// TIA Portal V19 export
TYPE "LAF_typeAxisDiagUnits"
TITLE = LAF_typeAxisDiagUnits
// Length and velocity units of a Technology Object
// stored: Access Published
   STRUCT
      lengthUnit { ExternalWritable := 'False'} : UDInt;   // Unit for position (1004=rad, 1005=°, 1010=m, 1011=km, 1013=mm, 1014=µm, 1015=nm, 1018=ft, 1019=in, 1021=mi); with high resolution (1536=mm, 1537=°)
      velocityUnit { ExternalWritable := 'False'} : UDInt;   // Unit for velocity (1061=m/s, 1062=mm/s, 1063=m/h 1064=km/h, 1066=in/s, 1067=ft/s, 1069=in/min, 1070=ft/min, 1075=mi/h, 1082=1/s, 1083=1/min, 1086=rad/s, 1521=°/s, 1522=°/min, 1523=rad/min, 1524=mm/min, 1525=m/min, 1526=mm/h, 1527=km/min, 1528=1/h); with high resolution (1538=mm/s, 1539=°/s) / Unit for velocity (1061=m/s, 1062=mm/s, 1063=m/h 1064=km/h, 1066=in/s, 1067=ft/s, 1069=in/min, 1070=ft/min, 1075=mi/h, 1082=1/s, 1083=1/min, 1086=rad/s, 1521=°/s, 1522=°/min, 1523=rad/min=1524: mm/min, 1525=m/min, 1526=mm/h, 1527=km/min, 1528=1/h); with high resolution (1538=mm/s, 1539=°/s)
   END_STRUCT;
END_TYPE
